RoboDK station: 03A - Basic Pick and Place.rdk

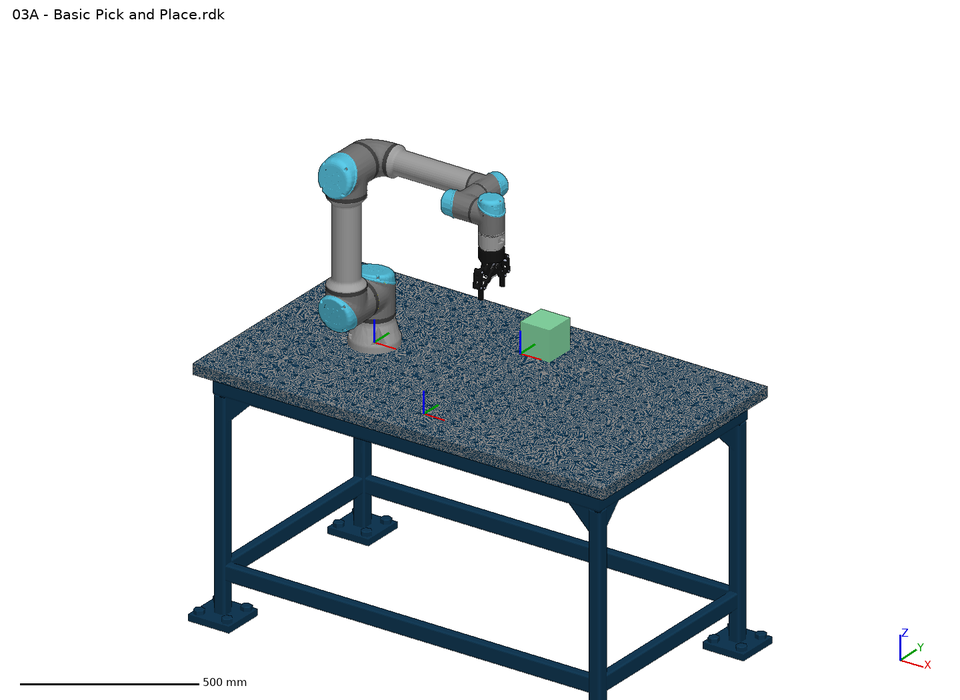
[picture v0: the station drawn from its stored meshes, robots at their saved joint values, targets as dots, program paths as lines]
Station 03A - Basic Pick and Place (saved by RoboDK 5.2.5). Poses are relative to the parent item; angles as X-Y-Z fixed-axis rotations.
Station parameters (name, value as stored): Palletizing Plugin
  - frame UR5e Base at (0, 0, 0) mm
    - robot UR5e: 6 axes, payload 5 kg, reach 850 mm, repeatability 0.03 mm, weight 18.4 kg
        modified DH rows (alpha deg, a mm, theta deg, d mm): 0, 0, 0, 162.5; 90, 0, 180, 0; 0, 425, 0, 0; 0, 392.25, 0, 133.3; -90, 0, 0, 99.7; 90, 0, 180, 99.6
        joint limits [-360, -360, -360, -360, -360, -360] to [360, 360, 360, 360, 360, 360]; home [0, -90, -90, -90, 90, 0]; saved at [0, -90, -90, -90, 90, 0]
      - tool Gripper RobotiQ 85 Opened, TCP at (0, 0, 130) mm, size 147.4 x 146.8 x 75 mm
  - frame World at (0, 0, 0) mm
    - object Table at (0, 0, 0) mm, size 1420 x 820 x 800 mm, geometry from Table-1400x800x800.sld
  - frame PositionA at (375, 175, 0) mm
    - object box at (50, 50, 50) mm, size 100 x 100 x 100 mm, geometry from box.sld
  - frame PositionB at (375, -295.45, 0) mm
